{attribute 'qualified_only'}
{attribute 'strict'}
TYPE E_TestStates :
(
    Unknown := 0,
    OUT := 1,
    TARGET1 := 2,
    TARGET2 := 3
) UINT;
END_TYPE

(* stored: Version 1.1.0.1
   DUT E_TestStates: Id {c258efcc-6b1f-486b-bdf8-0d1ba128e372} *)
